// TIA Portal V19 export
TYPE "C402_VAR_IF_M33_TYPIC"
   STRUCT
      STS_AAN { ExternalAccessible := 'False'; ExternalVisible := 'False'; ExternalWritable := 'False'} : Bool;   // TRUE = M33-bord actueel in werking FALSE = Uit
      EXT_AUT { ExternalAccessible := 'False'; ExternalVisible := 'False'; ExternalWritable := 'False'} : Bool;   // Externe (hoofd) beveiliging aangesproken
      EXT_HW { ExternalAccessible := 'False'; ExternalVisible := 'False'; ExternalWritable := 'False'} : Bool;   // Sturings hardware (PLC) in storing
      STO { ExternalAccessible := 'False'; ExternalVisible := 'False'; ExternalWritable := 'False'} : Struct   // Opsomming van alle storingen en meldingen
         A001 : Bool;   // Beveiliging aangesproken
         A002 : Bool;   // Storing M33-bord gedetecteerd door PRTG
         A003 : Bool;   // Storing M33-bord
         A004 : Bool;   // Algemene storing M33-bord
         AT01 : Bool;   // Foute terugmelding: M33-bord aangestuurd, terugmelding Aan niet (of te laat) ontvangen
         AT02 : Bool;   // Foute terugmelding: M33-bord niet aangestuurd, terugmelding Aan blijft aanwezig
      END_STRUCT;
   END_STRUCT;
END_TYPE
